# EPICS StreamDevice protocol: support/asyn4-33/asyn/makeSupport/streamSCPI/_NAME_Sup/dev_NAME_.proto
getIDN {
    out "*IDN?";
    in "%\$1[^\r\n]";
    ExtraInput = Ignore;
}

cmd {
    out "\$1";
}

setD {
    out "\$1 %d";
}
getD {
    out "\$1?";
    in "%d";
    ExtraInput = Ignore;
}
